INTERFACE ITF_BaseHMILoggerElement_View

(*			
	RafalOS
	Rafał Osajda		19.11.2025		TC 4024.66
	Czyści danych przy zmienia ramki po poprzedniej ramce
*)
METHOD PUBLIC ClearAfterScreen : BOOL
VAR_INPUT
END_VAR
END_METHOD

(*			
	EVERDE sp. z o.o.
	Rafał Osajda		09.09.2025		TC 4024.66
	Generuje tablicę zdarzeń dla podanego ID dla 0 dla wszystkich elementów
*)
METHOD PUBLIC GetEventTableForIDItem : BOOL
VAR_INPUT
	uiIdItem			: UINT;
END_VAR
END_METHOD

(*			
	EVERDE sp. z o.o.
	Rafał Osajda		09.09.2025		TC 4024.66
	Zwraca tablicę swoich zdarzeń
*)
METHOD PUBLIC GetYourEventTable : BOOL
VAR_INPUT
END_VAR
END_METHOD

(*			
	RafalOS
	Rafał Osajda		14.11.2025		TC 4024.66
	Metoda przygotowywania danych dla HMI 
	W niej odbywa się odpytywanie właściego elementu przez łącznik
*)
METHOD PUBLIC PrepareDataForHMI : BOOL
VAR_INPUT
END_VAR
END_METHOD

(*			
	RafalOS
	Rafał Osajda		19.11.2025		TC 4024.66
	Przygotowanie ramki pood tamke do wyświetlenia - tylko przygotowanie a nie przygotowanie danych do wyświetlenia
*)
METHOD PUBLIC PrepareForScreen : BOOL
VAR_INPUT
END_VAR
END_METHOD

END_INTERFACE

(* stored: Version 1.1.0.1
   Itf ITF_BaseHMILoggerElement_View: Id {5cb45a4d-d295-0879-1e7e-f79957b9c07c}
   Method ClearAfterScreen: Id {2177d0dc-fff4-07c6-039d-6d97b86c4606}
   Method GetEventTableForIDItem: Id {423d51d2-ec85-0a49-364c-a80a033c440a}
   Method GetYourEventTable: Id {df9a6c22-c1eb-0762-0f16-bbe7328d9649}
   Method PrepareDataForHMI: Id {634820b6-82e9-0625-1038-fe7e5f61cee9}
   Method PrepareForScreen: Id {63232c8c-3bcd-019c-111d-23e159556fed} *)
